Fanuc KAREL source: ka00002.KL

-- PROVISIONAL review KL for V770-1; original PC SHA256 a8bb52b786871f73dfddf4990822657eed7e5938d2758dbd23ab234593a4ec6f
-- Incomplete behavior may be omitted. Consult companion uncertainty JSON. Do not deploy.
PROGRAM KA00002
%NOLOCKGROUP
VAR
  SRC : INTEGER
  DST : REAL
BEGIN
  -- UNRESOLVED_PC offsets 5-16; opcodes 2E,23
  -- UNRESOLVED_PC offsets 21-34; opcodes 21,64,23
  -- UNRESOLVED_PC offsets 39-43; opcodes 7F
END KA00002
